(* IEC 61131-3 sources: Word/plc-course/02-electrical-and-field-devices/labs/starter, 3 files *)

(* ---- 02-1-fail-safe-motor.st ---- *)
(* Lab 02-1: Fail-safe motor circuit - NC stop and overload contacts.
   Module 02 (Electrical fundamentals and field devices).
   STARTER - the declarations are done for you; write the logic where it
   says TODO, then run:
     python3 tools/plctest.py 02-electrical-and-field-devices/labs/starter/02-1-fail-safe-motor.st
   Training exercise only: a real machine's emergency stop and safety
   functions are hard-wired or use safety-rated devices (Module 20). *)

PROGRAM FailSafeMotor
  VAR (* I/O - addresses follow the OpenPLC convention *)
    StartPB       AT %IX0.0 : BOOL;  (* Start push-button -S2, NO: TRUE while pressed *)
    StopPB_NC     AT %IX0.1 : BOOL;  (* Stop push-button -S1, NC: TRUE while NOT pressed *)
    OverloadOK_NC AT %IX0.2 : BOOL;  (* Overload relay -F2 contact 95-96, NC: TRUE while healthy *)
    Motor         AT %QX0.0 : BOOL;  (* Motor contactor -Q1 coil (through an interposing relay) *)
    TripLamp      AT %QX0.1 : BOOL;  (* Amber "overload tripped" lamp -H2 *)
  END_VAR

  (* TODO: replace these placeholder lines with your logic.
     Think about what each NC input reads when its wire breaks.
     (MATIEC needs at least one statement in a program body.) *)
  Motor := FALSE;
  TripLamp := FALSE;
END_PROGRAM

CONFIGURATION Config0
  RESOURCE Res0 ON PLC
    TASK MainTask(INTERVAL := T#10ms, PRIORITY := 0);
    PROGRAM Inst0 WITH MainTask : FailSafeMotor;
  END_RESOURCE
END_CONFIGURATION

(* ---- 02-2-solenoid-valves.st ---- *)
(* Lab 02-2: Solenoid valves - single-solenoid spring-return versus
   double-solenoid (bistable) valves on the same transfer line.
   Module 02 (Electrical fundamentals and field devices).
   STARTER - the declarations are done for you; write the logic where it
   says TODO, then run:
     python3 tools/plctest.py 02-electrical-and-field-devices/labs/starter/02-2-solenoid-valves.st
   Training exercise only: a real high-high level trip is a safety function
   and would be engineered separately (Module 20). *)

PROGRAM SolenoidValves
  VAR (* I/O - addresses follow the OpenPLC convention *)
    OpenPB         AT %IX0.0 : BOOL;  (* "Open line" push-button, NO: TRUE while pressed *)
    ClosePB_NC     AT %IX0.1 : BOOL;  (* "Close line" push-button, NC: TRUE while NOT pressed *)
    HighLevelOK_NC AT %IX0.2 : BOOL;  (* LSHH on the receiving tank, NC: TRUE while level is NOT high-high *)
    XV201_Sol      AT %QX0.0 : BOOL;  (* XV-201 solenoid: single-solenoid, spring return, fail closed *)
    XV202_OpenSol  AT %QX0.1 : BOOL;  (* XV-202 "open" coil: double-solenoid valve, stays put (fail last) *)
    XV202_CloseSol AT %QX0.2 : BOOL;  (* XV-202 "close" coil *)
  END_VAR
  VAR (* internal - add your own variables here if you need them *)
    Spare : BOOL;
  END_VAR

  (* TODO: replace these placeholder lines with your logic.
     The two valves receive the same commands but need different output
     patterns. What does each valve do when its coil is de-energised?
     (MATIEC needs at least one statement in a program body.) *)
  XV201_Sol := FALSE;
  XV202_OpenSol := FALSE;
  XV202_CloseSol := FALSE;
END_PROGRAM

CONFIGURATION Config0
  RESOURCE Res0 ON PLC
    TASK MainTask(INTERVAL := T#10ms, PRIORITY := 0);
    PROGRAM Inst0 WITH MainTask : SolenoidValves;
  END_RESOURCE
END_CONFIGURATION

(* ---- 02-3-namur-line-fault.st ---- *)
(* Lab 02-3: NAMUR sensor with line-fault detection - turn a switching
   signal plus open-circuit and short-circuit status bits into a validated
   signal and a fault.
   Module 02 (Electrical fundamentals and field devices).
   STARTER - the declarations are done for you; write the logic where it
   says TODO, then run:
     python3 tools/plctest.py 02-electrical-and-field-devices/labs/starter/02-3-namur-line-fault.st
   Training exercise only: this LSH is a control function. An independent
   high-high protection layer would be engineered separately (Module 20). *)

PROGRAM NamurLineFault
  VAR (* I/O - addresses follow the OpenPLC convention *)
    FillSel      AT %IX0.0 : BOOL;  (* Fill selector: TRUE = operator wants the tank filled *)
    SensorOn     AT %IX0.1 : BOOL;  (* LSH-301 via isolator: TRUE = NAMUR current in the ON band = fork dry *)
    WireBreak    AT %IX0.2 : BOOL;  (* Isolator status: open circuit detected (TRUE = fault) *)
    ShortCircuit AT %IX0.3 : BOOL;  (* Isolator status: short circuit detected (TRUE = fault) *)
    ResetPB      AT %IX0.4 : BOOL;  (* Fault reset push-button, NO: TRUE while pressed *)
    InletValve   AT %QX0.0 : BOOL;  (* XV-301 inlet valve solenoid, spring return: TRUE = open *)
    FaultLamp    AT %QX0.1 : BOOL;  (* Amber "LSH-301 line fault" lamp, latched *)
  END_VAR
  VAR (* internal - required by the lab interface *)
    LineFault : BOOL;  (* TRUE while an open or short circuit is present *)
    HighLevel : BOOL;  (* validated high level: TRUE when high OR when the signal cannot be trusted *)
  END_VAR

  (* TODO: replace these placeholder lines with your logic, in this order:
     LineFault, HighLevel, FaultLamp, InletValve.
     (MATIEC needs at least one statement in a program body.) *)
  LineFault := FALSE;
  HighLevel := FALSE;
  FaultLamp := FALSE;
  InletValve := FALSE;
END_PROGRAM

CONFIGURATION Config0
  RESOURCE Res0 ON PLC
    TASK MainTask(INTERVAL := T#10ms, PRIORITY := 0);
    PROGRAM Inst0 WITH MainTask : NamurLineFault;
  END_RESOURCE
END_CONFIGURATION
